FUNCTION_BLOCK FB_Visibilidad
VAR_INPUT
	Color 	 : DINT;
	Posicion : INT;
END_VAR
VAR_OUTPUT
END_VAR
VAR
END_VAR

IF Color = 1 THEN
	GVL.Clasificados[posicion-1].Visibilidad_Azul  := FALSE;	
	GVL.Clasificados[posicion-1].Visibilidad_Verde := TRUE;	
	GVL.Clasificados[posicion-1].Visibilidad_Metal := TRUE;			
	GVL.Clasificados[posicion-1].Visibilidad_Vacio := TRUE;	
ELSIF Color = 4 THEN
	GVL.Clasificados[posicion-1].Visibilidad_Azul  := TRUE;	
	GVL.Clasificados[posicion-1].Visibilidad_Verde := FALSE;	
	GVL.Clasificados[posicion-1].Visibilidad_Metal := TRUE;			
	GVL.Clasificados[posicion-1].Visibilidad_Vacio := TRUE;	
ELSIF Color = 7 THEN
	GVL.Clasificados[posicion-1].Visibilidad_Azul  := TRUE;	
	GVL.Clasificados[posicion-1].Visibilidad_Verde := TRUE;	
	GVL.Clasificados[posicion-1].Visibilidad_Metal := FALSE;			
	GVL.Clasificados[posicion-1].Visibilidad_Vacio := TRUE;	
ELSE
	GVL.Clasificados[posicion-1].Visibilidad_Azul  := TRUE;	
	GVL.Clasificados[posicion-1].Visibilidad_Verde := TRUE;	
	GVL.Clasificados[posicion-1].Visibilidad_Metal := TRUE;			
	GVL.Clasificados[posicion-1].Visibilidad_Vacio := FALSE;	
END_IF;

END_FUNCTION_BLOCK

(* stored: Version 1.1.0.1, ProductVersion 3.1.4024.12
   POU FB_Visibilidad: Id {7d48720f-99dc-4c71-bf0c-65d1fa0b8069}, SpecialFunc None *)
